(* IEC 61131-3 sources: beckhoffAutomationInterface/ST/Shark/Lib/BehaviorTree, 11 files *)

(* ---- E_CompareMode.st ---- *)
{attribute 'qualified_only'}
{attribute 'strict'}
TYPE E_CompareMode :
    (
        WITHIN_TOLERANCE := 0,
        GREATER_THAN := 1,
        LESS_THAN := 2
    ) DINT;
END_TYPE

(* ---- E_NodeStatus.st ---- *)
{attribute 'qualified_only'}
{attribute 'strict'}
TYPE E_NodeStatus :
    (
        IDLE := 0,
        RUNNING := 1,
        SUCCESS := 2,
        FAILURE := 3
    ) UDINT;
END_TYPE

(* ---- ST_NodeResult.st ---- *)
TYPE ST_NodeResult :
STRUCT
    eStatus       : E_NodeStatus;
    rProgress     : REAL;
    bHasError     : BOOL;
    stError       : ST_Error;        // Populated if bHasError = TRUE
    sDescription  : STRING(255);     // Human-readable status (e.g. "Step 2/4: Heating")
END_STRUCT
END_TYPE

(* ---- GVL_BT_Constants.st ---- *)
{attribute 'qualified_only'}
VAR_GLOBAL CONSTANT
    MAX_BT_CHILDREN : INT := 32;   // Max child nodes per container (Sequence, Parallel, etc.)
END_VAR

(* ---- I_TreeNode.st ---- *)
INTERFACE I_TreeNode
METHOD Tick : ST_NodeResult
END_METHOD

METHOD Reset : BOOL
END_METHOD

METHOD Halt
END_METHOD
END_INTERFACE

(* ---- F_BlendChildProgress.st ---- *)
(* F_BlendChildProgress - Blend a child node's progress with its index position
   inside an ordered composite (Sequence, ReactiveSequence).

   Returns overall progress 0..100 as:

       ((nChildIndex - 1) + rChildProgress / 100) / nTotalChildren * 100

   Guards against division by zero when nTotalChildren <= 0.
*)
FUNCTION F_BlendChildProgress : REAL
VAR_INPUT
    nChildIndex     : INT;  // 1-based index of the currently executing child
    nTotalChildren  : INT;  // total number of children in the composite
    rChildProgress  : REAL; // current child's progress, 0..100
END_VAR
    IF nTotalChildren <= 0 THEN
        F_BlendChildProgress := 0.0;
        RETURN;
    END_IF

    F_BlendChildProgress := (INT_TO_REAL(nChildIndex - 1) + rChildProgress / 100.0)
                           / INT_TO_REAL(nTotalChildren) * 100.0;
END_FUNCTION

(* ---- F_BuildNullChildResult.st ---- *)
(* F_BuildNullChildResult - Build a standard FAILURE result for an unconfigured
   child node on a behavior-tree decorator.

   Centralizes the null-child boilerplate that would otherwise be duplicated
   in every decorator node (Retry, Inverter, Timeout, Repeat, etc.).

   Usage inside a decorator's Tick method:

       IF _ipChild = 0 THEN
           Tick := F_BuildNullChildResult(sName, 'Xxx decorator child not configured');
           RETURN;
       END_IF
*)
FUNCTION F_BuildNullChildResult : ST_NodeResult
VAR_INPUT
    sSource  : STRING(80);
    sMessage : STRING(255);
END_VAR
    F_BuildNullChildResult.eStatus             := E_NodeStatus.FAILURE;
    F_BuildNullChildResult.bHasError           := TRUE;
    F_BuildNullChildResult.stError.eErrorId    := E_ErrorId.ERR_BT_NULL_CHILD;
    F_BuildNullChildResult.stError.sSource     := sSource;
    F_BuildNullChildResult.stError.sMessage    := sMessage;
END_FUNCTION

(* ---- F_BuildNullInterfaceResult.st ---- *)
(* F_BuildNullInterfaceResult - Build a standard FAILURE result for an unconfigured
   hardware interface on a behavior-tree leaf node.

   Centralizes the null-interface boilerplate that would otherwise be duplicated
   in every action node (OpenValve, CloseValve, SetController, etc.).

   Usage inside a node's Tick method:

       IF _ipValve = 0 THEN
           Tick := F_BuildNullInterfaceResult(sName, 'Valve interface not configured');
           RETURN;
       END_IF
*)
FUNCTION F_BuildNullInterfaceResult : ST_NodeResult
VAR_INPUT
    sSource  : STRING(80);
    sMessage : STRING(255);
END_VAR
    F_BuildNullInterfaceResult.eStatus             := E_NodeStatus.FAILURE;
    F_BuildNullInterfaceResult.bHasError           := TRUE;
    F_BuildNullInterfaceResult.stError.eErrorId    := E_ErrorId.ERR_BT_NULL_INTERFACE;
    F_BuildNullInterfaceResult.stError.sSource     := sSource;
    F_BuildNullInterfaceResult.stError.sMessage    := sMessage;
END_FUNCTION

(* ---- F_CompareModeToString.st ---- *)
(* F_CompareModeToString - Converts E_CompareMode to a human-readable string.
   Used in error messages and status descriptions (DRY). *)
FUNCTION F_CompareModeToString : STRING(20)
VAR_INPUT
    eMode : E_CompareMode;
END_VAR

    CASE eMode OF
        E_CompareMode.WITHIN_TOLERANCE:
        F_CompareModeToString := 'within';

        E_CompareMode.GREATER_THAN:
        F_CompareModeToString := '>';

        E_CompareMode.LESS_THAN:
        F_CompareModeToString := '<';
    ELSE
        F_CompareModeToString := '?';
    END_CASE
END_FUNCTION

(* ---- F_EvaluateCompareMode.st ---- *)
(* F_EvaluateCompareMode - Evaluates a value against a target using the specified compare mode.
   Centralizes comparison logic used by sensor action nodes (DRY). *)
FUNCTION F_EvaluateCompareMode : BOOL
VAR_INPUT
    rValue     : LREAL;
    rTarget    : LREAL;
    rTolerance : LREAL;         // Only used for WITHIN_TOLERANCE mode
    eMode      : E_CompareMode;
END_VAR

    CASE eMode OF
        E_CompareMode.WITHIN_TOLERANCE:
        F_EvaluateCompareMode := ABS(rValue - rTarget) <= rTolerance;

        E_CompareMode.GREATER_THAN:
        F_EvaluateCompareMode := rValue > rTarget;

        E_CompareMode.LESS_THAN:
        F_EvaluateCompareMode := rValue < rTarget;
    ELSE
        F_EvaluateCompareMode := FALSE;
    END_CASE
END_FUNCTION

(* ---- FB_Blackboard.st ---- *)
(* FB_Blackboard — Shared key-value store for Behavior Tree nodes

Provides a simple typed key-value store that nodes can use to share data.
Supports INT (DINT), REAL (LREAL), BOOL, and STRING types.
Keys are STRING(50). Max entries defined by constant.
*)
FUNCTION_BLOCK FB_Blackboard
VAR
    _asKeys    : ARRAY[1..MAX_ENTRIES] OF STRING(50);
    _anIntVals : ARRAY[1..MAX_ENTRIES] OF DINT;
    _arRealVals: ARRAY[1..MAX_ENTRIES] OF LREAL;
    _abBoolVals: ARRAY[1..MAX_ENTRIES] OF BOOL;
    _asStrVals : ARRAY[1..MAX_ENTRIES] OF STRING(255);
    _aeTypes   : ARRAY[1..MAX_ENTRIES] OF INT; // BB_TYPE_UNUSED=0, BB_TYPE_INT=1, BB_TYPE_REAL=2, BB_TYPE_BOOL=3, BB_TYPE_STRING=4
    _nCount    : INT := 0;
END_VAR
VAR CONSTANT
    MAX_ENTRIES    : INT := 64;
    BB_TYPE_UNUSED : INT := 0;
    BB_TYPE_INT    : INT := 1;
    BB_TYPE_REAL   : INT := 2;
    BB_TYPE_BOOL   : INT := 3;
    BB_TYPE_STRING : INT := 4;
END_VAR

METHOD PRIVATE _FindKey : INT
VAR_INPUT
    sKey : STRING(50);
END_VAR
VAR
    i : INT;
END_VAR
    FOR i := 1 TO _nCount DO
        IF _asKeys[i] = sKey THEN
            _FindKey := i;
            RETURN;
        END_IF
    END_FOR
    _FindKey := 0;
END_METHOD

METHOD PRIVATE _AllocKey : INT
VAR_INPUT
    sKey  : STRING(50);
    nType : INT;
END_VAR
VAR
    idx : INT;
END_VAR
    idx := _FindKey(sKey);
    IF idx > 0 THEN
        _aeTypes[idx] := nType;
        _AllocKey := idx;
        RETURN;
    END_IF

    IF _nCount >= MAX_ENTRIES THEN
        _AllocKey := 0;
        RETURN;
    END_IF

    _nCount := _nCount + 1;
    _asKeys[_nCount] := sKey;
    _aeTypes[_nCount] := nType;
    _AllocKey := _nCount;
END_METHOD

METHOD PUBLIC SetInt : BOOL
VAR_INPUT
    sKey   : STRING(50);
    nValue : DINT;
END_VAR
VAR
    idx : INT;
END_VAR
    idx := _AllocKey(sKey, BB_TYPE_INT);
    IF idx > 0 THEN
        _anIntVals[idx] := nValue;
        SetInt := TRUE;
    END_IF
END_METHOD

METHOD PUBLIC TryGetInt : BOOL
VAR_INPUT
    sKey : STRING(50);
END_VAR
VAR_OUTPUT
    nValue : DINT;
END_VAR
VAR
    idx : INT;
END_VAR
    idx := _FindKey(sKey);
    IF idx > 0 AND _aeTypes[idx] = BB_TYPE_INT THEN
        nValue := _anIntVals[idx];
        TryGetInt := TRUE;
    ELSE
        nValue := 0;
        TryGetInt := FALSE;
    END_IF
END_METHOD

METHOD PUBLIC SetReal : BOOL
VAR_INPUT
    sKey   : STRING(50);
    rValue : LREAL;
END_VAR
VAR
    idx : INT;
END_VAR
    idx := _AllocKey(sKey, BB_TYPE_REAL);
    IF idx > 0 THEN
        _arRealVals[idx] := rValue;
        SetReal := TRUE;
    END_IF
END_METHOD

METHOD PUBLIC TryGetReal : BOOL
VAR_INPUT
    sKey : STRING(50);
END_VAR
VAR_OUTPUT
    rValue : LREAL;
END_VAR
VAR
    idx : INT;
END_VAR
    idx := _FindKey(sKey);
    IF idx > 0 AND _aeTypes[idx] = BB_TYPE_REAL THEN
        rValue := _arRealVals[idx];
        TryGetReal := TRUE;
    ELSE
        rValue := 0.0;
        TryGetReal := FALSE;
    END_IF
END_METHOD

METHOD PUBLIC SetBool : BOOL
VAR_INPUT
    sKey   : STRING(50);
    bValue : BOOL;
END_VAR
VAR
    idx : INT;
END_VAR
    idx := _AllocKey(sKey, BB_TYPE_BOOL);
    IF idx > 0 THEN
        _abBoolVals[idx] := bValue;
        SetBool := TRUE;
    END_IF
END_METHOD

METHOD PUBLIC TryGetBool : BOOL
VAR_INPUT
    sKey : STRING(50);
END_VAR
VAR_OUTPUT
    bValue : BOOL;
END_VAR
VAR
    idx : INT;
END_VAR
    idx := _FindKey(sKey);
    IF idx > 0 AND _aeTypes[idx] = BB_TYPE_BOOL THEN
        bValue := _abBoolVals[idx];
        TryGetBool := TRUE;
    ELSE
        bValue := FALSE;
        TryGetBool := FALSE;
    END_IF
END_METHOD

METHOD PUBLIC SetString : BOOL
VAR_INPUT
    sKey   : STRING(50);
    sValue : STRING(255);
END_VAR
VAR
    idx : INT;
END_VAR
    idx := _AllocKey(sKey, BB_TYPE_STRING);
    IF idx > 0 THEN
        _asStrVals[idx] := sValue;
        SetString := TRUE;
    END_IF
END_METHOD

METHOD PUBLIC TryGetString : BOOL
VAR_INPUT
    sKey : STRING(50);
END_VAR
VAR_OUTPUT
    sValue : STRING(255);
END_VAR
VAR
    idx : INT;
END_VAR
    idx := _FindKey(sKey);
    IF idx > 0 AND _aeTypes[idx] = BB_TYPE_STRING THEN
        sValue := _asStrVals[idx];
        TryGetString := TRUE;
    ELSE
        sValue := '';
        TryGetString := FALSE;
    END_IF
END_METHOD

END_FUNCTION_BLOCK
